FUNCTION_BLOCK fbVerwarming
VAR_INPUT
	bDrukknop				:BOOL;
	bThermostaat			:BOOL;
	bVerlichting			:BOOL;
	tTijdVoorStart			:TIME;
END_VAR
VAR_OUTPUT
	bKlep_open				:BOOL;
	bBrander				:BOOL;
END_VAR
VAR
	bUitlooptijdKlep			:BOOL;
	Uitlooptijd					:tof;
	TijdsduurVoorverwarming		:tof;
	Brander						:F_TRIG;
	
END_VAR

TijdsduurVoorverwarming(IN:= bDrukknop, PT:= tTijdVoorStart, Q=> , ET=> );

Uitlooptijd(IN:= bUitlooptijdKlep, PT:= T#30S, Q=> , ET=> );

IF Uitlooptijd.Q THEN
	bKlep_open := TRUE;
	ELSE
	bKlep_open := FALSE;
	END_IF

IF (TijdsduurVoorverwarming.Q OR bVerlichting) AND bThermostaat THEN
		bUitlooptijdKlep := TRUE;
		bBrander := TRUE;
		ELSE
		bUitlooptijdKlep :=FALSE;
		bBrander := FALSE;
END_IF

END_FUNCTION_BLOCK

(* stored: Version 1.1.0.1, ProductVersion 3.1.4024.12
   POU fbVerwarming: Id {373aaa5f-de6f-4177-8425-08ce9f094437}, SpecialFunc None *)
